// TIA Portal V16 export
// export: Created 2025-10-06T17:54:39.2133206Z, ExportSetting WithDefaults, DisplayName Totally Integrated Automation Portal, DisplayVersion V16, DisplayName TIA Portal Version Control Interface, DisplayVersion V16, DisplayName TIA Portal Openness, DisplayVersion V16, DisplayName STEP 7 Professional, DisplayVersion V16, DisplayName STEP 7 Safety, DisplayVersion V16, DisplayName WinCC Advanced, DisplayVersion V16
DATA_BLOCK "Override_Block_Safety_1"   // DB3
VERSION : 0.1
// stored: AutoNumber true, InstanceOfName Override_Block_Safety, InstanceOfType FB
"Override_Block_Safety"
   // VAR_INPUT
   //    "SAFE Q 1" : Bool;
   //    "SAFE Q 2" : Bool;
   //    "Override Contact" : Bool;
   //    "Delay Timer" : Time;
   // END_VAR
   // VAR_OUTPUT
   //    "SAFE Output Contact" : Bool;
   //    "Timer ET" : Time;
   // END_VAR
BEGIN
END_DATA_BLOCK
